// Block: PPrgArchive18

DATA_BLOCK PPrgArchive18
VERSION : 0.1
   NON_RETAIN
   VAR
      PRG : Array[1701..1800] of PPrg_Data;
   END_VAR

BEGIN
   // No initialization required
END_DATA_BLOCK
